Fanuc KAREL source: kb00095.KL

-- PROVISIONAL review KL for V770-1; original PC SHA256 9beedc059f57b78e9a9eeb2c951cf6a2e4a4bc3aa7644ab848817f5177c5bc39
-- Incomplete behavior may be omitted. Consult companion uncertainty JSON. Do not deploy.
PROGRAM KB00095
%NOLOCKGROUP
BEGIN
  -- UNRESOLVED_PC offsets 5-12; opcodes 9D,23
  -- UNRESOLVED_PC offsets 17-24; opcodes 9D,23
  -- UNRESOLVED_PC offsets 29-38; opcodes 3F,75
  -- UNRESOLVED_PC offsets 43-50; opcodes 9D,23
  -- UNRESOLVED_PC offsets 55-85; opcodes 27,22,22,22,2A,22,31
  -- UNRESOLVED_PC offsets 90-94; opcodes 7F
END KB00095
